PROGRAM MAIN
VAR
END_VAR

END_PROGRAM

(* stored: Version 1.1.0.1
   POU MAIN: Id {33c727ef-2466-4aa6-b7f7-fb22e88db091} *)
